PROGRAM MAIN
VAR
	udiDeviceID 			: UDINT 	:= 1;
	sTargetNetID 			: STRING 	:= '192.168.1.20.1.1';
	sSlaveDescriptionPath	: STRING 	:= 'C:\TwinCAT\3.1\Config\Io\EtherCAT';
	udiZoomFactor 			: UDINT 	:= 3;
	bReadOnly 				: BOOL;
	bSowSlaveInfo			: BOOL;
	bShowOnlineTopology		: BOOL;
	bRefresh 				: BOOL;
	
END_VAR

;

END_PROGRAM

(* stored: Version 1.1.0.1, ProductVersion 3.1.4024.3
   POU MAIN: Id {50b8efee-224c-4311-8177-06af3dcc3016}, SpecialFunc None *)
